// TIA Portal project "Project1" (V18)

(* hardware
DEVICE "S7-1500/ET200MP station_1"  S7-1500 station
   slot 0: "Rail_0"  Rack  6ES7 590-1***0-0AA0
   slot 1: "PLC_1"  CPU 1518-4 PN/DP  6ES7 518-4AP00-0AB0  V3.0
      slot 3: "CPU display_1"  6ES7591-1BA00-0AA0
      slot 32768: "PROFINET interface_1"  X1
         slot 32769: "Port_1"  X1 P1
         slot 32770: "Port_2"  X1 P2
      slot 33024: "PROFINET interface_2"  X2
         slot 33025: "Port_1"  X2 P1
      slot 33280: "PROFINET interface GBIT_3"  X3
         slot 33281: "Port_1"  X3 P1
      slot 33536: "DP interface_1"  X4
      slot 34817: "Virtual CP interface port_1"  Virtual CP interface port  Virtual CP interface port
*)

// ===== PLC "PLC_1"  CPU 1518-4 PN/DP =====

VAR_GLOBAL   // PLC tag table "Default tag table"
   "Tag_1" AT %I0.0 : Bool;
   "Tag_2" AT %I0.1 : Bool;
   "Tag_3" AT %I0.2 : Bool;
   "Tag_4" AT %QW0 : Word;
END_VAR

DATA_BLOCK "FB_10_DB"   // DB1
{ S7_Optimized_Access := 'TRUE' }
VERSION : 0.1
// stored: InstanceOfName FB_10
"FB_10"
BEGIN
END_DATA_BLOCK

FUNCTION_BLOCK "FB_01"   // FB1, LAD
TITLE = ON_MODE
{ S7_Optimized_Access := 'TRUE' }
VERSION : 0.1
   VAR_INPUT
      ST_SP : Bool;
   END_VAR
   VAR_OUTPUT
      ON_MODE : Bool;
   END_VAR
   VAR
      K1 : Bool;
      P1 : Bool;
      RDY : Bool;
   END_VAR
   VAR_TEMP   // added for the SCL form of the ladder/FBD networks
      _w1 : Bool;
   END_VAR
BEGIN

REGION Network 1: 입력 신호를 상승 펄스 신호 출력으로 변환
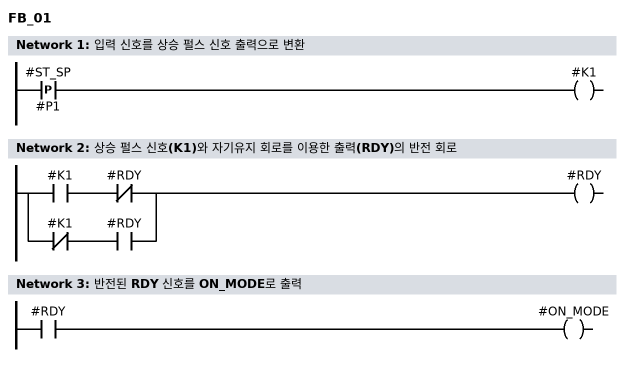
   RUNG wire#powerrail
      P_Contact(operand := #ST_SP, bit := #P1)
      Coil( #K1 )
   END_RUNG
   // the same network as SCL:
   #_w1 := #ST_SP AND NOT #P1;   // rising edge of #ST_SP
   #P1 := #ST_SP;
   #K1 := #_w1;
END_REGION

REGION Network 2: 상승 펄스 신호(K1)와 자기유지 회로를 이용한 출력(RDY)의 반전 회로
   RUNG wire#powerrail
      Contact( #K1 )
      I_Contact( #RDY )
      wire#w1
      Coil( #RDY )
   END_RUNG
   RUNG wire#powerrail
      I_Contact( #K1 )
      Contact( #RDY )
   END_RUNG wire#w1
   // the same network as SCL:
   #RDY := (#K1 AND NOT #RDY) OR (NOT #K1 AND #RDY);
END_REGION

REGION Network 3: 반전된 RDY 신호를 ON_MODE로 출력
   RUNG wire#powerrail
      Contact( #RDY )
      Coil( #ON_MODE )
   END_RUNG
   // the same network as SCL:
   #ON_MODE := #RDY;
END_REGION
END_FUNCTION_BLOCK

FUNCTION_BLOCK "FB_02"   // FB2, LAD
TITLE = ON - INC & DEC
{ S7_Optimized_Access := 'TRUE' }
VERSION : 0.1
   VAR_INPUT
      ON_IN : Bool;
      UP_PB : Bool;
      DN_PB : Bool;
   END_VAR
   VAR_OUTPUT
      I_CNT_OUT : Int;
   END_VAR
   VAR
      I_PB_CNT : Int;
      P1 : Bool;
      P2 : Bool;
      P3 : Bool;
      P4 : Bool;
   END_VAR
   VAR_TEMP   // added for the SCL form of the ladder/FBD networks
      _w1 : Bool;
      _w2 : Bool;
   END_VAR
BEGIN

REGION Network 1: 전원 버튼이 눌러져 전원이 ON될 때 FND모듈에 숫자 1을 표시
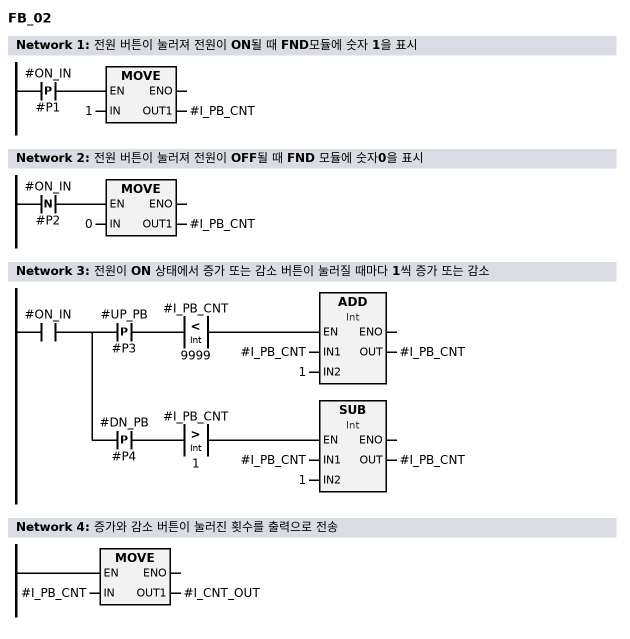
   RUNG wire#powerrail
      P_Contact(operand := #ON_IN, bit := #P1)
      Move(in := 1, out1 => #I_PB_CNT)
   END_RUNG
   // the same network as SCL:
   #_w1 := #ON_IN AND NOT #P1;   // rising edge of #ON_IN
   #P1 := #ON_IN;
   IF #_w1 THEN #I_PB_CNT := 1; END_IF;
END_REGION

REGION Network 2: 전원 버튼이 눌러져 전원이 OFF될 때 FND 모듈에 숫자0을 표시
   RUNG wire#powerrail
      N_Contact(operand := #ON_IN, bit := #P2)
      Move(in := 0, out1 => #I_PB_CNT)
   END_RUNG
   // the same network as SCL:
   #_w1 := NOT #ON_IN AND #P2;   // falling edge of #ON_IN
   #P2 := #ON_IN;
   IF #_w1 THEN #I_PB_CNT := 0; END_IF;
END_REGION

REGION Network 3: 전원이 ON 상태에서 증가 또는 감소 버튼이 눌러질 때마다 1씩 증가 또는 감소
   RUNG wire#powerrail
      Contact( #ON_IN )
      wire#w1
      P_Contact(operand := #UP_PB, bit := #P3)
      { S7_Templates := "SrcType := Int" } LT_Contact(in1 := #I_PB_CNT, in2 := 9999)
      { S7_Templates := "SrcType := Int" } Add(in1 := #I_PB_CNT, in2 := 1, out => #I_PB_CNT)
   END_RUNG
   RUNG wire#w1
      P_Contact(operand := #DN_PB, bit := #P4)
      { S7_Templates := "SrcType := Int" } GT_Contact(in1 := #I_PB_CNT, in2 := 1)
      { S7_Templates := "SrcType := Int" } Sub(in1 := #I_PB_CNT, in2 := 1, out => #I_PB_CNT)
   END_RUNG
   // the same network as SCL:
   #_w1 := #ON_IN AND #UP_PB AND NOT #P3;   // rising edge of #UP_PB
   #P3 := #UP_PB;
   IF #_w1 AND (#I_PB_CNT < 9999) THEN #I_PB_CNT := #I_PB_CNT + 1; END_IF;
   #_w2 := #ON_IN AND #DN_PB AND NOT #P4;   // rising edge of #DN_PB
   #P4 := #DN_PB;
   IF #_w2 AND (#I_PB_CNT > 1) THEN #I_PB_CNT := #I_PB_CNT - 1; END_IF;
END_REGION

REGION Network 4: 증가와 감소 버튼이 눌러진 횟수를 출력으로 전송
   RUNG wire#powerrail
      Move(in := #I_PB_CNT, out1 => #I_CNT_OUT)
   END_RUNG
   // the same network as SCL:
   #I_CNT_OUT := #I_PB_CNT;
END_REGION
END_FUNCTION_BLOCK

FUNCTION_BLOCK "FB_10"   // FB3, LAD
{ S7_Optimized_Access := 'TRUE' }
VERSION : 0.1
   VAR_INPUT
      ST_SP : Bool;
      UP_PB : Bool;
      DN_PB : Bool;
   END_VAR
   VAR_OUTPUT
      W_FND_OUT : Word;
   END_VAR
   VAR
      ON_STATE : Bool;
      I_CNT_TEMP : Int;
      FB_01_Instance : "FB_01";
      FB_02_Instance : "FB_02";
   END_VAR
BEGIN

REGION Network 1: OB1에서 FB_01을 호출
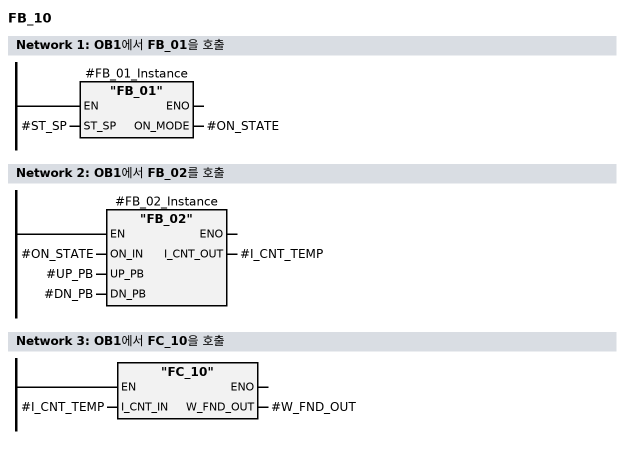
   RUNG wire#powerrail
      #FB_01_Instance(ST_SP := #ST_SP, ON_MODE => #ON_STATE)
   END_RUNG
   // the same network as SCL:
   #FB_01_Instance(ST_SP := #ST_SP, ON_MODE => #ON_STATE);   // "FB_01"
END_REGION

REGION Network 2: OB1에서 FB_02를 호출
   RUNG wire#powerrail
      #FB_02_Instance(ON_IN := #ON_STATE, UP_PB := #UP_PB, DN_PB := #DN_PB, I_CNT_OUT => #I_CNT_TEMP)
   END_RUNG
   // the same network as SCL:
   #FB_02_Instance(ON_IN := #ON_STATE, UP_PB := #UP_PB, DN_PB := #DN_PB, I_CNT_OUT => #I_CNT_TEMP);   // "FB_02"
END_REGION

REGION Network 3: OB1에서 FC_10을 호출
   RUNG wire#powerrail
      "FC_10"(I_CNT_IN := #I_CNT_TEMP, W_FND_OUT => #W_FND_OUT)
   END_RUNG
   // the same network as SCL:
   "FC_10"(I_CNT_IN := #I_CNT_TEMP, W_FND_OUT => #W_FND_OUT);
END_REGION
END_FUNCTION_BLOCK

FUNCTION "FC_01" : Void   // FC1, LAD
{ S7_Optimized_Access := 'TRUE' }
VERSION : 0.1
   VAR_INPUT
      I_CNT_IN : Int;
   END_VAR
   VAR_OUTPUT
      W_BCD_OUT : Word;
   END_VAR
   VAR_TEMP
      D_CNT_DI : DInt;
      D_CNT_BCD : DWord;
   END_VAR
BEGIN

REGION Network 1: INT형을 DINT형으로 변환 후에 정수값을 BCD코드로 변환
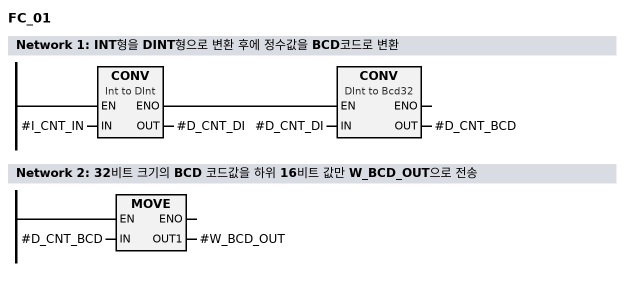
   RUNG wire#powerrail
      { S7_Templates := "[SrcType := Int, DestType := DInt]" } Convert(in := #I_CNT_IN, out => #D_CNT_DI)
      { S7_Templates := "[SrcType := DInt, DestType := Bcd32]" } Convert(in := #D_CNT_DI, out => #D_CNT_BCD)
   END_RUNG
   // the same network as SCL:
   #D_CNT_DI := INT_TO_DINT(#I_CNT_IN);
   #D_CNT_BCD := DINT_TO_BCD32(#D_CNT_DI);
END_REGION

REGION Network 2: 32비트 크기의 BCD 코드값을 하위 16비트 값만 W_BCD_OUT으로 전송
   RUNG wire#powerrail
      Move(in := #D_CNT_BCD, out1 => #W_BCD_OUT)
   END_RUNG
   // the same network as SCL:
   #W_BCD_OUT := #D_CNT_BCD;
END_REGION
END_FUNCTION

FUNCTION "FC_02" : Void   // FC2, STL
{ S7_Optimized_Access := 'TRUE' }
VERSION : 0.1
   VAR_INPUT
      W_BCD_IN : Word;
   END_VAR
   VAR_OUTPUT
      W_FND_OUT : Word;
   END_VAR
BEGIN

REGION Network 1: 빅 엔디안 방식의 BCD 코드를 입력 받아서 리틀 엔디안 방식으로 변경
         L     #W_BCD_IN;
         CAW;
         T     #W_FND_OUT;
END_REGION
END_FUNCTION

FUNCTION "FC_03" : Void   // FC3, LAD
{ S7_Optimized_Access := 'TRUE' }
VERSION : 0.1
   VAR_INPUT
      W_BCD_IN : Word;
   END_VAR
   VAR_OUTPUT
      W_FND_OUT : Word;
   END_VAR
   VAR_TEMP
      W_BCD_SHL : Word;
      W_BCD_SHR : Word;
   END_VAR
BEGIN

REGION Network 1: STL로 작성한 CAW명령어와 같은 기능을 한다.
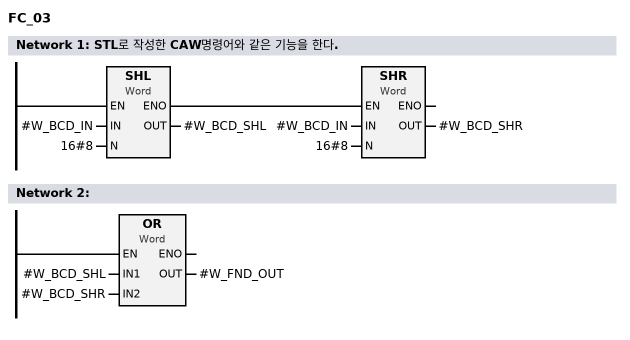
   RUNG wire#powerrail
      { S7_Templates := "SrcType := Word" } Shl(in := #W_BCD_IN, n := 16#8, out => #W_BCD_SHL)
      { S7_Templates := "SrcType := Word" } Shr(in := #W_BCD_IN, n := 16#8, out => #W_BCD_SHR)
   END_RUNG
   // the same network as SCL:
   #W_BCD_SHL := SHL(IN := #W_BCD_IN, N := 16#8);
   #W_BCD_SHR := SHR(IN := #W_BCD_IN, N := 16#8);
END_REGION

REGION Network 2
   #W_FND_OUT := #W_BCD_SHL OR #W_BCD_SHR;
END_REGION
END_FUNCTION

FUNCTION "FC_10" : Void   // FC4, LAD
{ S7_Optimized_Access := 'TRUE' }
VERSION : 0.1
   VAR_INPUT
      I_CNT_IN : Int;
   END_VAR
   VAR_OUTPUT
      W_FND_OUT : Word;
   END_VAR
   VAR_TEMP
      W_BCD_TEMP : Word;
   END_VAR
BEGIN

REGION Network 1: I_CNT_IN의 정수값을 BCD 코드로 변환하는 블록 호출
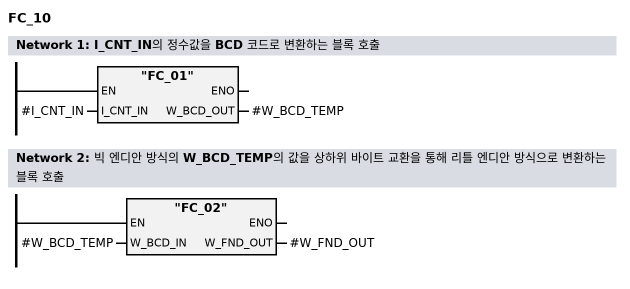
   RUNG wire#powerrail
      "FC_01"(I_CNT_IN := #I_CNT_IN, W_BCD_OUT => #W_BCD_TEMP)
   END_RUNG
   // the same network as SCL:
   "FC_01"(I_CNT_IN := #I_CNT_IN, W_BCD_OUT => #W_BCD_TEMP);
END_REGION

REGION Network 2: 빅 엔디안 방식의 W_BCD_TEMP의 값을 상하위 바이트 교환을 통해 리틀 엔디안 방식으로 변환하는 블록 호출
   RUNG wire#powerrail
      "FC_02"(W_BCD_IN := #W_BCD_TEMP, W_FND_OUT => #W_FND_OUT)
   END_RUNG
   // the same network as SCL:
   "FC_02"(W_BCD_IN := #W_BCD_TEMP, W_FND_OUT => #W_FND_OUT);
END_REGION
END_FUNCTION

ORGANIZATION_BLOCK "Main"   // OB1, LAD, ProgramCycle
TITLE = "Main Program Sweep (Cycle)"
{ S7_Optimized_Access := 'TRUE' }
VERSION : 0.1
   VAR_INPUT
      Initial_Call : Bool;   // Initial call of this OB
      Remanence : Bool;   // =True, if remanent data are available
   END_VAR
BEGIN

REGION Network 1
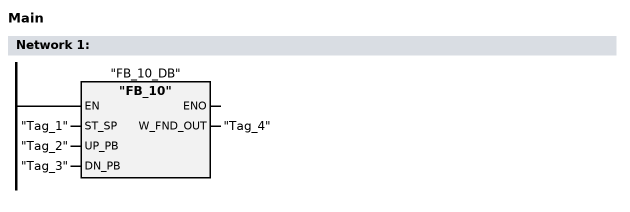
   RUNG wire#powerrail
      "FB_10_DB"(ST_SP := "Tag_1", UP_PB := "Tag_2", DN_PB := "Tag_3", W_FND_OUT => "Tag_4")
   END_RUNG
   // the same network as SCL:
   "FB_10_DB"(ST_SP := "Tag_1", UP_PB := "Tag_2", DN_PB := "Tag_3", W_FND_OUT => "Tag_4");   // "FB_10"
END_REGION
END_ORGANIZATION_BLOCK